{attribute 'qualified_only'}
VAR_GLOBAL
 DI: ARRAY[0..1023] OF BYTE;
END_VAR

(* stored: Version 1.1.0.1, ProductVersion 3.1.4024.5
   GVL DigInput: Id {1be1f3ce-5170-42d0-8978-48d2e2665a48} *)
